{attribute 'GeneratedUsingTerminal: KL8524'}
{attribute addProperty BoxType "KL8524"}
{attribute addProperty Description ""}
{attribute addProperty Physics ""}
{attribute addProperty Id "Channel_1AT %Q*Channel_3263D8D50"}
{attribute addProperty CRC "2763596142"}
{attribute addProperty Size "0"}
TYPE KL8524_A4B9216E :
STRUCT
	{attribute addProperty Name "Channel_1"}
	Channel_1 : Channel_3263D8D5;
END_STRUCT
END_TYPE

(* stored: Version 1.2.0.0, ProductVersion 3.1.4024.9
   DUT KL8524_A4B9216E: Id {4ed33348-4c1b-481f-8bb1-727e89713042} *)
